# EPICS substitutions: src/iocdoc/testfiles/iocBoot/ioc495idc/templates/placeholders.substitutions
file "$(TOP)/495idcApp/Db/phAnalogout.db"
{
pattern
{P	H	F		D}
# NPI
{495idc:	sft01:	ph01:	ao01 }
{495idc:	sft01:	ph01:	ao02 }
{495idc:	sft01:	ph01:	ao03 }
{495idc:	sft01:	ph01:	ao04 }
{495idc:	sft01:	ph01:	ao05 }
{495idc:	sft01:	ph01:	ao06 }
{495idc:	sft01:	ph01:	ao07 }
{495idc:	sft01:	ph01:	ao08 }
{495idc:	sft01:	ph01:	ao09 }
{495idc:	sft01:	ph01:	ao10 }
{495idc:	sft01:	ph01:	ao11 }
{495idc:	sft01:	ph01:	ao12 }
{495idc:	sft01:	ph01:	ao13 }
{495idc:	sft01:	ph01:	ao14 }
{495idc:	sft01:	ph01:	ao15 }
{495idc:	sft01:	ph01:	ao16 }
{495idc:	sft01:	ph01:	ao17 }
{495idc:	sft01:	ph01:	ao18 }
{495idc:	sft01:	ph01:	ao19 }
{495idc:	sft01:	ph01:	ao20 }
# DET
{495idc:	sft01:	ph02:	ao01 }
{495idc:	sft01:	ph02:	ao02 }
{495idc:	sft01:	ph02:	ao03 }
{495idc:	sft01:	ph02:	ao04 }
{495idc:	sft01:	ph02:	ao05 }
{495idc:	sft01:	ph02:	ao06 }
{495idc:	sft01:	ph02:	ao07 }
{495idc:	sft01:	ph02:	ao08 }
{495idc:	sft01:	ph02:	ao09 }
{495idc:	sft01:	ph02:	ao10 }
{495idc:	sft01:	ph02:	ao11 }
{495idc:	sft01:	ph02:	ao12 }
{495idc:	sft01:	ph02:	ao13 }
{495idc:	sft01:	ph02:	ao14 }
{495idc:	sft01:	ph02:	ao15 }
{495idc:	sft01:	ph02:	ao16 }
{495idc:	sft01:	ph02:	ao17 }
{495idc:	sft01:	ph02:	ao18 }
{495idc:	sft01:	ph02:	ao19 }
{495idc:	sft01:	ph02:	ao20 }
# NES
{495idc:	sft01:	ph03:	ao01 }
{495idc:	sft01:	ph03:	ao02 }
{495idc:	sft01:	ph03:	ao03 }
{495idc:	sft01:	ph03:	ao04 }
{495idc:	sft01:	ph03:	ao05 }
{495idc:	sft01:	ph03:	ao06 }
{495idc:	sft01:	ph03:	ao07 }
{495idc:	sft01:	ph03:	ao08 }
{495idc:	sft01:	ph03:	ao09 }
{495idc:	sft01:	ph03:	ao10 }
{495idc:	sft01:	ph03:	ao11 }
{495idc:	sft01:	ph03:	ao12 }
{495idc:	sft01:	ph03:	ao13 }
{495idc:	sft01:	ph03:	ao14 }
{495idc:	sft01:	ph03:	ao15 }
{495idc:	sft01:	ph03:	ao16 }
{495idc:	sft01:	ph03:	ao17 }
{495idc:	sft01:	ph03:	ao18 }
{495idc:	sft01:	ph03:	ao19 }
{495idc:	sft01:	ph03:	ao20 }

}

file "$(TOP)/495idcApp/Db/phBinaryout.db"
{
pattern
{P	H	F	D	MSK	ON	OFF}

{495idc:	sft01:	ph01:	bo01	0x00001	"On"	"Off" }
{495idc:	sft01:	ph01:	bo02	0x00002	"On"	"Off" }
{495idc:	sft01:	ph01:	bo03	0x00004	"On"	"Off" }
{495idc:	sft01:	ph01:	bo04	0x00008	"On"	"Off" }
{495idc:	sft01:	ph01:	bo05	0x00010	"On"	"Off" }
{495idc:	sft01:	ph01:	bo06	0x00020	"On"	"Off" }
{495idc:	sft01:	ph01:	bo07	0x00040	"On"	"Off" }
{495idc:	sft01:	ph01:	bo08	0x00080	"On"	"Off" }
{495idc:	sft01:	ph01:	bo09	0x00100	"On"	"Off" }
{495idc:	sft01:	ph01:	bo10	0x00200	"On"	"Off" }
{495idc:	sft01:	ph01:	bo11	0x00400	"On"	"Off" }
{495idc:	sft01:	ph01:	bo12	0x00800	"On"	"Off" }
{495idc:	sft01:	ph01:	bo13	0x01000	"On"	"Off" }
{495idc:	sft01:	ph01:	bo14	0x02000	"On"	"Off" }
{495idc:	sft01:	ph01:	bo15	0x04000	"On"	"Off" }
{495idc:	sft01:	ph01:	bo16	0x08000	"On"	"Off" }
{495idc:	sft01:	ph01:	bo17	0x10000	"On"	"Off" }
{495idc:	sft01:	ph01:	bo18	0x20000	"On"	"Off" }
{495idc:	sft01:	ph01:	bo19	0x40000	"On"	"Off" }
{495idc:	sft01:	ph01:	bo20	0x80000	"On"	"Off" }

}

file "$(TOP)/495idcApp/Db/phLongout.db"
{
pattern
{P	H	F	D}
# NES
{495idc:	sft01:	ph01:	lo01 }
{495idc:	sft01:	ph01:	lo02 }
{495idc:	sft01:	ph01:	lo03 }
{495idc:	sft01:	ph01:	lo04 }
{495idc:	sft01:	ph01:	lo05 }
{495idc:	sft01:	ph01:	lo06 }
{495idc:	sft01:	ph01:	lo07 }
{495idc:	sft01:	ph01:	lo08 }
{495idc:	sft01:	ph01:	lo09 }
{495idc:	sft01:	ph01:	lo10 }
{495idc:	sft01:	ph01:	lo11 }
{495idc:	sft01:	ph01:	lo12 }
{495idc:	sft01:	ph01:	lo13 }
{495idc:	sft01:	ph01:	lo14 }
{495idc:	sft01:	ph01:	lo15 }
{495idc:	sft01:	ph01:	lo16 }
{495idc:	sft01:	ph01:	lo17 }
{495idc:	sft01:	ph01:	lo18 }
{495idc:	sft01:	ph01:	lo19 }
{495idc:	sft01:	ph01:	lo20 }

}

file "$(TOP)/495idcApp/Db/phStringout.db"
{
pattern
{P	H	F	D}

{495idc:	sft01:	ph01:	so01 }
{495idc:	sft01:	ph01:	so02 }
{495idc:	sft01:	ph01:	so03 }
{495idc:	sft01:	ph01:	so04 }
{495idc:	sft01:	ph01:	so05 }
{495idc:	sft01:	ph01:	so06 }
{495idc:	sft01:	ph01:	so07 }
{495idc:	sft01:	ph01:	so08 }
{495idc:	sft01:	ph01:	so09 }
{495idc:	sft01:	ph01:	so10 }
{495idc:	sft01:	ph01:	so11 }
{495idc:	sft01:	ph01:	so12 }
{495idc:	sft01:	ph01:	so13 }
{495idc:	sft01:	ph01:	so14 }
{495idc:	sft01:	ph01:	so15 }
{495idc:	sft01:	ph01:	so16 }
{495idc:	sft01:	ph01:	so17 }
{495idc:	sft01:	ph01:	so18 }
{495idc:	sft01:	ph01:	so19 }
{495idc:	sft01:	ph01:	so20 }

}
